FUNCTION_BLOCK Process
VAR_INPUT
	Rob: FB_Robot;
	Fleet: FB_Robot;
	CNC: FB_CNC;

END_VAR


	

VAR_OUTPUT
END_VAR
VAR
	bExecute: BOOL;
END_VAR

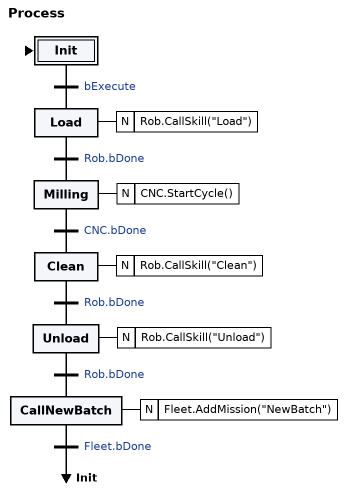
INITIAL_STEP Init:
END_STEP
TRANSITION FROM Init TO Load
    := bExecute;
END_TRANSITION
STEP Load:
    Rob.CallSkill("Load")(N);
END_STEP
TRANSITION FROM Load TO Milling
    := Rob.bDone;
END_TRANSITION
STEP Milling:
    CNC.StartCycle()(N);
END_STEP
TRANSITION FROM Milling TO Clean
    := CNC.bDone;
END_TRANSITION
STEP Clean:
    Rob.CallSkill("Clean")(N);
END_STEP
TRANSITION FROM Clean TO Unload
    := Rob.bDone;
END_TRANSITION
STEP Unload:
    Rob.CallSkill("Unload")(N);
END_STEP
TRANSITION FROM Unload TO CallNewBatch
    := Rob.bDone;
END_TRANSITION
STEP CallNewBatch:
    Fleet.AddMission("NewBatch")(N);
END_STEP
TRANSITION FROM CallNewBatch TO Init
    := Fleet.bDone;
END_TRANSITION

END_FUNCTION_BLOCK

(* stored: Version 1.1.0.1, ProductVersion 3.1.4026.18
   POU Process: Id {95e2959f-04b0-4bba-b119-5c97b4077463}, SpecialFunc None *)
